// TIA Portal V20 export
TYPE "LWONIK_typeZoneStatus"
// stored: Access Published
   STRUCT
      safetyReleased1 : Bool;
      safetyReleased2 : Bool;
      safetyReleased3 : Bool;
      safetyReleased4 : Bool;
      ackReq : Bool;
      safetyFault : Bool;
      highSpeedEnable : Bool;
      activeSLS { ExternalWritable := 'False'} : Bool;   // SLS is activated on Zone
      activeSTO { ExternalWritable := 'False'} : Bool;   // STO is activated on Zone
      activeSOS { ExternalWritable := 'False'} : Bool;   // STO is activated on Zone
      activeSS1 { ExternalWritable := 'False'} : Bool;   // STO is activated on Zone
      activeSS2 { ExternalWritable := 'False'} : Bool;   // STO is activated on Zone
      AllFDoorClose : Bool;   // All Door Close
      SFDoorOpen : Bool;
      MFDoorOpen : Bool;
   END_STRUCT;
END_TYPE
